{attribute 'linkalways'} 
{attribute 'no_explicit_call' := 'This FB is a CLASS and must be accessed using methods or properties'}
{attribute 'enable_dynamic_creation'}
FUNCTION_BLOCK AsyncCommand IMPLEMENTS I_AsyncCommand
VAR
	stateMachine : AsyncCommandStateMachine;
END_VAR

METHOD PUBLIC Abort
VAR_INPUT
END_VAR
stateMachine.Abort();
END_METHOD

PROPERTY PUBLIC Busy : BOOL
GET
IF stateMachine.IsAborted THEN
	RETURN;
END_IF

IF stateMachine.IsCompleted THEN
	RETURN;
END_IF

IF stateMachine.IsErrored THEN
	RETURN;
END_IF

IF stateMachine.IsIdle THEN
	RETURN;
END_IF

Busy := TRUE;
END_GET
END_PROPERTY

METHOD PUBLIC CyclicCall
VAR_INPUT
END_VAR
IF stateMachine.IsIdle THEN
	OnIdle();
END_IF

IF stateMachine.IsInitializing THEN
	OnInitializing(stateMachine);
END_IF

IF stateMachine.IsExecuting THEN
	OnExecuting(stateMachine);
END_IF

IF stateMachine.IsCompleting THEN
	OnCompleting(stateMachine);
END_IF

IF stateMachine.IsCompleted THEN
	OnCompleted();
END_IF

IF stateMachine.IsAborting THEN
	OnAborting(stateMachine);
END_IF

IF stateMachine.IsAborted THEN
	OnAborted();
END_IF

IF stateMachine.IsErrored THEN
	OnErrored();
END_IF
END_METHOD

PROPERTY PUBLIC Done : BOOL
GET
Done := stateMachine.IsCompleted;
END_GET
END_PROPERTY

PROPERTY PUBLIC Error : BOOL
GET
Error := stateMachine.IsErrored;
END_GET
END_PROPERTY

PROPERTY PUBLIC ErrorId : UDINT
GET
ErrorId := stateMachine.ErrorId;
END_GET
END_PROPERTY

METHOD PUBLIC Execute
VAR_INPUT
END_VAR
stateMachine.Execute();
END_METHOD

METHOD PROTECTED OnAborted
VAR_INPUT
END_VAR
END_METHOD

METHOD PROTECTED OnAborting
VAR_INPUT
	StateControl : I_AsyncCommandStateControl;
END_VAR
// default behaviour is to go to next state
// you can override this method to implement your own completing control code.
// just call StateControl.Next() when your code is completed.  

StateControl.Next();
END_METHOD

METHOD PROTECTED OnCompleted : BOOL
VAR_INPUT
END_VAR
END_METHOD

METHOD PROTECTED OnCompleting
VAR_INPUT
	StateControl : I_AsyncCommandStateControl;
END_VAR
// default behaviour is to go to next state
// you can override this method to implement your own completing control code.
// just call StateControl.Next() when your code is completed.  

StateControl.Next();
END_METHOD

METHOD PROTECTED OnErrored
VAR_INPUT
END_VAR
END_METHOD

METHOD PROTECTED OnExecuting
VAR_INPUT
	StateControl : I_AsyncCommandStateControl;
END_VAR
// default behaviour is to go to next state
// you can override this method to implement your own executing control code.
// just call StateControl.Next() when your code is completed.  

StateControl.Next();
END_METHOD

METHOD PROTECTED OnIdle
VAR_INPUT
END_VAR
END_METHOD

METHOD PROTECTED OnInitializing
VAR_INPUT
	StateControl : I_AsyncCommandStateControl;
END_VAR
// default behaviour is to go to next state
// you can override this method to implement your own initializing control code.
// just call StateControl.Next() when your code is completed.  

StateControl.Next();
END_METHOD

END_FUNCTION_BLOCK

(* stored: Version 1.1.0.1, ProductVersion 3.1.4024.12
   POU AsyncCommand: Id {167a49ad-66b7-036c-12b3-201b18025f30}, SpecialFunc None
   Folder Protected: Id {85307ef1-af44-0248-0fab-eb879ad107a4}
   Method Abort: Id {a0ee3453-a67e-0d75-280d-16ca0de9e3b1}
   Property Busy: Id {9ef4397e-5594-0537-0a97-14aa93a4b51f}
   Get Get: Id {8ff75693-55a4-0918-396a-e0523dbf2cb9}
   Method CyclicCall: Id {6854302e-2920-05d4-24af-826647146430}
   Property Done: Id {35c23c46-e1fc-0546-16c3-7c66a4ba5a6c}
   Get Get: Id {e8a22a7e-9cb1-0654-0f52-fdeb969fe48e}
   Property Error: Id {94fff5aa-c6ee-0c58-344c-3f4b723a0921}
   Get Get: Id {cb991754-6eeb-047b-14ac-9efdf04f7e5f}
   Property ErrorId: Id {2bd8c94b-c57f-031c-0729-2c59968d082e}
   Get Get: Id {47b50b14-0a76-0cdd-0e94-791454875457}
   Method Execute: Id {9ef3fabe-0a17-09db-0297-faa6903e2cb3}
   Method OnAborted: Id {a161191a-5171-07e1-1d26-555c3baaff8a}
   Method OnAborting: Id {d7fd0d33-b736-0547-1fd6-5341b5070afe}
   Method OnCompleted: Id {f38d45e0-70e2-040a-3005-476f66428176}
   Method OnCompleting: Id {d1957dcc-5026-0772-2ab8-861a5a1a286d}
   Method OnErrored: Id {e957eb3f-db39-0428-0e38-d504ae4abc07}
   Method OnExecuting: Id {b0592078-a554-0fb1-1f2a-ed2aaf25ec2f}
   Method OnIdle: Id {617bed85-8a96-0694-0a4b-23410e7e287a}
   Method OnInitializing: Id {96172a5e-3643-0b54-2a1a-aef3ad07f4b4} *)
